TYPE ST_LaudaReadCommands_ActuatingSignal :
STRUCT
	Value	: STRING := 'IN_PV_06';
END_STRUCT
END_TYPE

(* stored: Version 1.1.0.1, ProductVersion 3.1.4024.12
   DUT ST_LaudaReadCommands_ActuatingSignal: Id {3d2004aa-a7ae-4dc2-956f-c1941b38022a} *)
